FUNCTION_BLOCK Seq_Ausrichten_MPlate EXTENDS FB_Basis IMPLEMENTS I_Sequenz
VAR_INPUT
	// Skillzuweisung
	R_Move					:I_Skill_RoboterErweitert;
	G_Move					:I_Skill_SmartGreifer;
	
	// Prozessparameter		
	RobParam				:ARRAY[0..4] OF sRoboterProzessVariablen;
	GripParam				:sSmartGreiferProzessVariablen;
	ErreichtParam			:sKraftVariablen;
END_VAR
VAR_OUTPUT
END_VAR
VAR
	// Interne Sequenzen
	Seq_Ausrichten			:Seq_Ausrichten;	

	// Interne Paramater 
	Ausrichten_Pos			:ARRAY[0..1] OF sRoboterProzessVariablen;
	ErreichtParamReset		:sKraftVariablen;
END_VAR

// Ablauf
ACT_Ablauf();

// Zustandshandling
CASE iState OF
	0:	// BEREIT
		IF bStart THEN
			iState := 1;
		END_IF
	1:	// LAUFEND
		IF eSysCommand = 4 THEN
			bReset := TRUE;
			SFCReset := TRUE;
		END_IF
		
		IF bBeendet OR bReset THEN
			bReset := FALSE;
			SFCReset := FALSE;
			iState := 0;
		END_IF
	2: // ABGESCHLOSSEN
		IF SFCCurrentStep = 'Init' THEN
			iState := 0;
		END_IF
END_CASE

ACTION ACT_Ablauf:
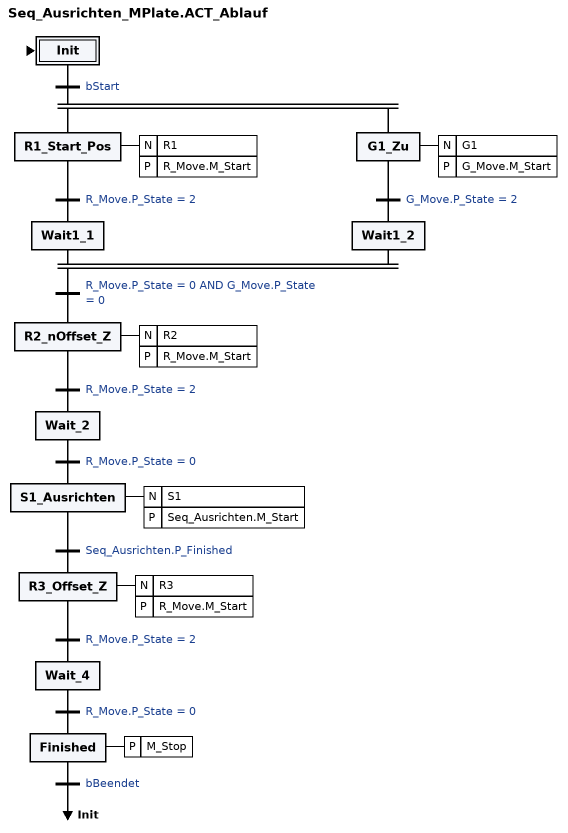
INITIAL_STEP Init:
END_STEP
TRANSITION FROM Init TO (R1_Start_Pos, G1_Zu)
    := bStart;
END_TRANSITION
STEP R1_Start_Pos:
    R1(N);
    R_Move.M_Start(P);
END_STEP
TRANSITION FROM R1_Start_Pos TO Wait1_1
    := R_Move.P_State = 2;
END_TRANSITION
STEP Wait1_1:
END_STEP
STEP G1_Zu:
    G1(N);
    G_Move.M_Start(P);
END_STEP
TRANSITION FROM G1_Zu TO Wait1_2
    := G_Move.P_State = 2;
END_TRANSITION
STEP Wait1_2:
END_STEP
TRANSITION FROM (Wait1_1, Wait1_2) TO R2_nOffset_Z
    := R_Move.P_State = 0 AND G_Move.P_State = 0;
END_TRANSITION
STEP R2_nOffset_Z:
    R2(N);
    R_Move.M_Start(P);
END_STEP
TRANSITION FROM R2_nOffset_Z TO Wait_2
    := R_Move.P_State = 2;
END_TRANSITION
STEP Wait_2:
END_STEP
TRANSITION FROM Wait_2 TO S1_Ausrichten
    := R_Move.P_State = 0;
END_TRANSITION
STEP S1_Ausrichten:
    S1(N);
    Seq_Ausrichten.M_Start(P);
END_STEP
TRANSITION FROM S1_Ausrichten TO R3_Offset_Z
    := Seq_Ausrichten.P_Finished;
END_TRANSITION
STEP R3_Offset_Z:
    R3(N);
    R_Move.M_Start(P);
END_STEP
TRANSITION FROM R3_Offset_Z TO Wait_4
    := R_Move.P_State = 2;
END_TRANSITION
STEP Wait_4:
END_STEP
TRANSITION FROM Wait_4 TO Finished
    := R_Move.P_State = 0;
END_TRANSITION
STEP Finished:
    M_Stop(P);
END_STEP
TRANSITION FROM Finished TO Init
    := bBeendet;
END_TRANSITION
END_ACTION

ACTION G1:
G_Move.P_SGripperParam := GripParam;
END_ACTION

ACTION R1:
R_Move.P_RobotParam := RobParam[0];
END_ACTION

ACTION R2:
R_Move.P_RobotParam := RobParam[1];
END_ACTION

ACTION R3:
R_Move.P_RobotParam := RobParam[4];
END_ACTION

ACTION S1:
Ausrichten_Pos[0] := RobParam[2];
Ausrichten_Pos[1] := RobParam[3];

Seq_Ausrichten(	eSysCommand := GVL.SystemCommand,
				R_Move := SkillSet.Move_2P2_Advanced,
				RobParam := Ausrichten_Pos,
				ErreichtParam := ErreichtParam);
END_ACTION

END_FUNCTION_BLOCK

(* stored: Version 1.1.0.1
   POU Seq_Ausrichten_MPlate: Id {aa0a329e-1383-4fc8-a7ba-ba7cada9e1dd}, SpecialFunc None
   Folder 01_Zuweisung: Id {3c37cb1c-75de-45c0-bae5-d7c1201c9aa4}
   Action ACT_Ablauf: Id {62e931ce-4889-4fd6-8793-516eb185be1b}
   Action G1: Id {796ee13a-6770-4428-8a91-187977221775}
   Action R1: Id {9e703a3f-5d85-48ff-b0b4-c083ef3c9a33}
   Action R2: Id {58019613-0f7b-4638-a369-f9ee31c45971}
   Action R3: Id {025121c3-2dfb-449f-9048-c06e78b51f2f}
   Action S1: Id {0b362b00-eb52-4c68-b5b2-594863508356} *)
